// TwinCAT 3 PLC project StringsTests
// ProgramVersion: 3.1.4024.0
// libraries:
//   Strings, * (TomasRompotl)
//   Tc2_Standard, * (Beckhoff Automation GmbH)
//   Tc2_System, * (Beckhoff Automation GmbH)
//   Tc3_Module, * (Beckhoff Automation GmbH)
//   TcUnit, * (www.tcunit.org)
//   Types, * (TomasRompotl)
// project tree:
//   / PlcTask.TcTTO
//   Tests/Builders/ StringBuilder255Test.TcPOU, BuildStringInlineTest.TcPOU, StringBuilderExtBufferTest.TcPOU, StringBuilderInfiniteTest.TcPOU
//   Tests/Convert/ ConvertFunctionsTest.TcPOU
//   Tests/Manipulate/ ManipulateFunctionsTest.TcPOU
//   Tests/ PRG_Test.TcPOU
//   Tests/Validate/ ValidateFunctionsTest.TcPOU
//   Tests/_TemplateTest/ _TemplateTest.TcPOU
// (motion and I/O tree: see PLC project types)
// real-time tasks:
//   TASK BindingTestTask: cycle T#10ms, priority 20, ADS port 350
//   TASK PlcTask: cycle T#10ms, priority 21, ADS port 351
//   TASK PlcTask1: cycle T#10ms, priority 22, ADS port 352
//   TASK PlcTask2: cycle T#10ms, priority 23, ADS port 353

CONFIGURATION StringsTests
    RESOURCE PLC ON TwinCAT3
        TASK PlcTask(INTERVAL := T#1ms, PRIORITY := 21);
        PROGRAM PRG_Test WITH PlcTask : PRG_Test;
    END_RESOURCE
END_CONFIGURATION

// ---- Tests/PRG_Test.TcPOU
PROGRAM PRG_Test
VAR
	validateFunctionsTest : ValidateFunctionsTest;
	manipulateFunctionsTest : ManipulateFunctionsTest;
	convertFunctionsTest : ConvertFunctionsTest;
	
	sb255Test : StringBuilder255Test;
	buildStringInlineTest : BuildStringInlineTest;
	sbExtBufferTest : StringBuilderExtBufferTest;
	sbInfiniteTest : StringBuilderInfiniteTest;
END_VAR

TcUnit.RUN();

END_PROGRAM

// ---- Tests/Validate/ValidateFunctionsTest.TcPOU
FUNCTION_BLOCK ValidateFunctionsTest EXTENDS TcUnit.FB_TestSuite
VAR
END_VAR

StringBeginsWithAnyFunction();
StringEndsWithAnyFunction();
StringBeginsWithFunction();
StringEndsWithFunction();

METHOD StringBeginsWithAnyFunction : BOOL
VAR
	test : T_MaxString := 'this is test string';
END_VAR
TcUnit.TEST('String begins with');

AssertEquals_BOOL(
	Expected := FALSE,
	Actual := StringBeginsWithAny(test, 'nothing'),
	Message := 'Should return FALSE because string does not begin with checked value');

AssertEquals_BOOL(
	Expected := TRUE,
	Actual := StringBeginsWithAny(test, 'this'),
	Message := 'Should return TRUE because string begins with checked value');

TEST_FINISHED();
END_METHOD

METHOD StringBeginsWithFunction
VAR
	test : T_MaxString := 'this is test string';
END_VAR
TcUnit.TEST('String begins with function');

AssertEquals_BOOL(
	Expected := FALSE,
	Actual := StringBeginsWith(test, 'nothing'),
	Message := 'Should return FALSE because string does not begin with checked value');

AssertEquals_BOOL(
	Expected := TRUE,
	Actual := StringBeginsWith(test, 'this'),
	Message := 'Should return TRUE because string begins with checked value');

TEST_FINISHED();
END_METHOD

METHOD StringEndsWithAnyFunction : BOOL
VAR
	test : T_MaxString := 'this is test string';
END_VAR
TcUnit.TEST('String ends with');

AssertEquals_BOOL(
	Expected := FALSE,
	Actual := StringBeginsWithAny(test, 'nothing'),
	Message := 'Should return FALSE because string does not end with checked value');

AssertEquals_BOOL(
	Expected := TRUE,
	Actual := StringEndsWithAny(test, 'string'),
	Message := 'Should return TRUE because string ends with checked value');

TEST_FINISHED();
END_METHOD

METHOD StringEndsWithFunction
VAR
	test : T_MaxString := 'this is test string';
END_VAR
TcUnit.TEST('String ends with function');

AssertEquals_BOOL(
	Expected := FALSE,
	Actual := StringBeginsWith(test, 'nothing'),
	Message := 'Should return FALSE because string does not end with checked value');

AssertEquals_BOOL(
	Expected := TRUE,
	Actual := StringEndsWith(test, 'string'),
	Message := 'Should return TRUE because string ends with checked value');

TEST_FINISHED();
END_METHOD

END_FUNCTION_BLOCK

// ---- Tests/Manipulate/ManipulateFunctionsTest.TcPOU
FUNCTION_BLOCK ManipulateFunctionsTest EXTENDS TcUnit.FB_TestSuite
VAR
END_VAR

AddLeadingZerosFunction();
GetStringBetweenFunction();
RemoveStringFromEndFunction();
ReplaceStringFunction();
ReplaceAllFunction();
ReplaceAllAnyFunction();
ReplaceAllAnyTypeFunction();
SubstringFunction();

METHOD AddLeadingZerosFunction : BOOL
VAR
	test : T_MaxString := '555';
END_VAR
TcUnit.TEST('Add leading zeros');

AssertEquals_STRING(
	Expected := '00555',
	Actual := AddLeadingZeros(test, 5),
	Message := 'Should pad propper number of zeros');

AssertEquals_STRING(
	Expected := '555',
	Actual := AddLeadingZeros(test, 2),
	Message := 'Should do nothing if formatter string already has more chars');

TEST_FINISHED();
END_METHOD

METHOD GetStringBetweenFunction : BOOL
VAR
	test0 : T_MaxString := '1';
	test1 : T_MaxString := '[2]';
	test2 : T_MaxString := 'TestValue[3]rest';
	actual : T_MaxString;
END_VAR
TcUnit.TEST('Get string between');

actual := GetStringBetween(test0, '[', ']');

AssertEquals_STRING(
	Expected := '',
	Actual := actual,
	Message := 'Should return nothing');

actual := GetStringBetween(test1, '[', ']');

AssertEquals_STRING(
	Expected := '2',
	Actual := actual,
	Message := 'Should return content of brackets');

actual := GetStringBetween(test2, '[', ']');

AssertEquals_STRING(
	Expected := '3',
	Actual := actual,
	Message := 'Should return content of brackets');

TEST_FINISHED();
END_METHOD

METHOD RemoveStringFromEndFunction : BOOL
VAR
	test : T_MaxString := 'Last word will be removed';
	actual : T_MaxString;
END_VAR
TcUnit.TEST('Remove string from end function');

actual := RemoveStringFromEnd(test, 'removed');

AssertEquals_STRING(
	Expected := 'Last word will be ',
	Actual := actual,
	Message := 'Should remove last word from test string');

TEST_FINISHED();
END_METHOD

METHOD ReplaceAllAnyFunction
VAR  
	inputString : T_MaxString := 'Valve1 is open';
	substringToReplace : T_MaxString := 'Valve1'; 
	replacementSubstring : T_MaxString := 'Valve2';
 
END_VAR
TcUnit.TEST('Replace all any function');  

ReplaceAllAny(inputString, substringToReplace, replacementSubstring); 

AssertEquals_STRING(
	Expected := 'Valve2 is open',
	Actual := inputString,
	Message := 'Should delete the substring if replacement is empty');
	
TEST_FINISHED();
END_METHOD

METHOD ReplaceAllAnyTypeFunction
VAR  
	inputString  : T_MaxString; 
	substringToReplace : T_MaxString;
	replacementSubstring : T_MaxString;
END_VAR
TcUnit.TEST('Replace all any type function');

inputString  := 'Valve1 is open';
substringToReplace := 'Valve1';
replacementSubstring  := 'Valve2';

ReplaceAllAnyType(ToAnyType(inputString), substringToReplace, replacementSubstring); 

AssertEquals_STRING(
	Expected := 'Valve2 is open',
	Actual := inputString,
	Message := 'ReplaceAllAnyType should delete the substring if replacement is empty');
	
inputString  := 'Valve1 is open';
substringToReplace := 'Valve4';
replacementSubstring  := 'Valve2';

ReplaceAllAnyType(ToAnyType(inputString), substringToReplace, replacementSubstring); 

AssertEquals_STRING(
	Expected := 'Valve1 is open',
	Actual := inputString,
	Message := 'ReplaceAllAnyType should not modify the string if no match is found');
	
inputString  := 'Valve1 is open';
substringToReplace := 'Valve1';
replacementSubstring  := '';

ReplaceAllAnyType(ToAnyType(inputString), substringToReplace, replacementSubstring);

AssertEquals_STRING(
	Expected := ' is open',
	Actual := inputString,
	Message := 'ReplaceAllAnyType should delete the substring if replacement is empty');
	
inputString  := 'Valve1 is open. Valve1 is closed';
substringToReplace := 'Valve1';
replacementSubstring  := 'V1';

ReplaceAllAnyType(ToAnyType(inputString), substringToReplace, replacementSubstring);

AssertEquals_STRING(
	Expected := 'V1 is open. V1 is closed',
	Actual := inputString,
	Message := 'ReplaceAllAnyType should replace all occurrences of the target text');

TEST_FINISHED();
END_METHOD

METHOD ReplaceAllFunction
VAR
	inputString  : T_MaxString;
	substringToReplace : T_MaxString;
	replacementSubstring  : T_MaxString;
END_VAR
TcUnit.TEST('Replace all function');

inputString  := 'Valve1 is open';
substringToReplace := 'Valve1';
replacementSubstring  := 'Valve2';
 
AssertEquals_STRING(
	Expected := 'Valve2 is open',
	Actual := ReplaceAll(inputString, substringToReplace, replacementSubstring),
	Message := 'ReplaceAll should correctly replace the target substring in the input string');
	
inputString  := 'Valve1 is open';
substringToReplace := 'Valve4';
replacementSubstring  := 'Valve2';

AssertEquals_STRING(
	Expected := 'Valve1 is open',
	Actual := ReplaceAll(inputString, substringToReplace, replacementSubstring),
	Message := 'Should not modify the string if no match is found');
	
inputString  := 'Valve1 is open';
substringToReplace := 'Valve1';
replacementSubstring  := '';

AssertEquals_STRING(
	Expected := ' is open',
	Actual := ReplaceAll(inputString, substringToReplace, replacementSubstring),
	Message := 'Should delete the substring if replacement is empty');
	
inputString  := 'Valve1 is open. Valve1 is closed';
substringToReplace := 'Valve1';
replacementSubstring  := 'V1';

AssertEquals_STRING(
	Expected := 'V1 is open. V1 is closed',
	Actual := ReplaceAll(inputString, substringToReplace, replacementSubstring),
	Message := 'ReplaceAll should replace all occurrences of the target text');

TEST_FINISHED();
END_METHOD

METHOD ReplaceStringFunction : BOOL
VAR
	test : T_MaxString := 'this is test string';
END_VAR
TcUnit.TEST('Replace string');

ReplaceString(test, 'not here', 'replaced');

AssertEquals_STRING(
	Expected := 'this is test string',
	Actual := test,
	Message := 'Should do nothing because searched string is not there');

ReplaceString(test, 'test', 'replaced');

AssertEquals_STRING(
	Expected := 'this is replaced string',
	Actual := test,
	Message := 'Should replace found string');

TEST_FINISHED();
END_METHOD

METHOD SubstringFunction
VAR
	source : T_MaxString :=  'ABCDEF123456789';
	destination : T_MaxString;
	startIndex : DINT := 3; 
    length : DINT := 5;	  
END_VAR
TcUnit.TEST('SubString function');

SubString(source, destination, startIndex, length);
AssertEquals_STRING(Expected := 'DEF12',
					Actual :=  destination, 
					Message := 'Substring result incorrect');

TEST_FINISHED();
END_METHOD

END_FUNCTION_BLOCK

// ---- Tests/Convert/ConvertFunctionsTest.TcPOU
FUNCTION_BLOCK ConvertFunctionsTest EXTENDS TcUnit.FB_TestSuite
VAR
END_VAR

AnyToStringFunction();
StringToAnyFunction();

METHOD AnyToStringFunction : BOOL
VAR
	stringVar : T_MaxString := 'test';
	intVar : INT := 42;
	realVar : REAL := 3.14;
END_VAR
TcUnit.TEST('ANY to STRING function');

AssertEquals_STRING(
	Expected := 'test',
	Actual := AnyToString(stringVar),
	Message := 'Should convert STRING var to STRING');

AssertEquals_STRING(
	Expected := '42',
	Actual := AnyToString(intVar),
	Message := 'Should convert INT var to STRING');

AssertEquals_STRING(
	Expected := '3.14',
	Actual := AnyToString(realVar),
	Message := 'Should convert REAL var to STRING');
	
TEST_FINISHED();
END_METHOD

METHOD StringToAnyFunction : BOOL
VAR
	stringVar : T_MaxString;
	intVar : INT;
	realVar : REAL;
END_VAR
TcUnit.TEST('STRING to ANY function');

StringToAny('this is test', stringVar);
StringToAny('42', intVar);
StringToAny('3.14', realVar);

AssertEquals_STRING(
	Expected := 'this is test',
	Actual := stringVar,
	Message := 'Should return correct STRING value');

AssertEquals_INT(
	Expected := 42,
	Actual := intVar,
	Message := 'Should return correct INT value');

AssertEquals_REAL(
	Expected := 3.14,
	Actual := realVar,
	Delta := 0.001,
	Message := 'Should return correct REAL value');

TEST_FINISHED();
END_METHOD

END_FUNCTION_BLOCK

// ---- Tests/Builders/StringBuilder255Test.TcPOU
FUNCTION_BLOCK StringBuilder255Test EXTENDS TcUnit.FB_TestSuite
VAR
END_VAR

AppendAndClear();

METHOD AppendAndClear : BOOL
VAR
	builder : StringBuilder255;
END_VAR
TcUnit.TEST('Append and Clear');

builder
	.Clear()
	.Append('1')
	.Append('2');

AssertEquals_STRING(
	Expected := '12',
	Actual := builder.GetString(),
	Message := 'Should return Appended strings using GetString() method');

AssertEquals_STRING(
	Expected := '12',
	Actual := builder.Value,
	Message := 'Should return string using Value property');

AssertEquals_DINT(
	Expected := 2,
	Actual := builder.Length,
	Message := 'Should return string length');	

builder.Clear();

AssertEquals_BOOL(
	Expected := TRUE,
	Actual := builder.IsEmpty,
	Message := 'Should return that string is empty');
	
TEST_FINISHED();
END_METHOD

END_FUNCTION_BLOCK

// ---- Tests/Builders/BuildStringInlineTest.TcPOU
FUNCTION_BLOCK BuildStringInlineTest EXTENDS TcUnit.FB_TestSuite
VAR
END_VAR

BuildStringInSingleLine();

METHOD BuildStringInSingleLine : BOOL
VAR
END_VAR
TcUnit.TEST('Build string in single line');

AssertEquals_STRING(
	Expected := '12',
	Actual := BuildStringInline('1').Append('2').GetString(),
	Message := 'Should return built string');

AssertEquals_STRING(
	Expected := 'ab',
	Actual := BuildStringInline('a').Append('b').GetString(),
	Message := 'Should return another built string');

TEST_FINISHED();
END_METHOD

END_FUNCTION_BLOCK

// ---- Tests/Builders/StringBuilderExtBufferTest.TcPOU
FUNCTION_BLOCK StringBuilderExtBufferTest EXTENDS TcUnit.FB_TestSuite
VAR
END_VAR

AppendAndClear();

METHOD AppendAndClear : BOOL
VAR
	buffer : STRING(2000);
	builder : StringBuilderExtBuffer := (Buffer := ToAnyType(buffer));
	
	testValue : STRING := ' very long strings';
END_VAR
TcUnit.TEST('Append and Clear');

builder
	.Clear()
	.Append('SB with external buffer')
	.Append(' is meant for')
	.AppendByPointer(ADR(testValue));

AssertEquals_STRING(
	Expected := 'SB with external buffer is meant for very long strings',
	Actual := buffer,
	Message := 'Strings should be properly appended');

builder.Clear();

AssertEquals_BOOL(
	Expected := TRUE,
	Actual := builder.IsEmpty,
	Message := 'Buffer should be empty');
	
TEST_FINISHED();
END_METHOD

END_FUNCTION_BLOCK

// ---- Tests/Builders/StringBuilderInfiniteTest.TcPOU
FUNCTION_BLOCK StringBuilderInfiniteTest EXTENDS TcUnit.FB_TestSuite
VAR
END_VAR

AppendAndClear();
CheckCapacityHasIncreased();

METHOD AppendAndClear : BOOL
VAR
	builder : StringBuilderInfinite;
	testValue : STRING := ' very long strings without care';
END_VAR
TcUnit.TEST('Append and Clear');

builder
	.Clear()
	.Append('SB infinite')
	.Append(' is meant for')
	.AppendByPointer(ADR(testValue));

AssertEquals_STRING(
	Expected := 'SB infinite is meant for very long strings without care',
	Actual := builder.Value^,
	Message := 'Strings should be properly appended');

builder.Clear();

AssertEquals_BOOL(
	Expected := TRUE,
	Actual := builder.IsEmpty,
	Message := 'String should be empty');
	
TEST_FINISHED();
END_METHOD

METHOD CheckCapacityHasIncreased : BOOL
VAR
	builder : StringBuilderInfinite;
	i : INT;
END_VAR
TcUnit.TEST('Check capacity has increased');

AssertEquals_DINT(
	Expected := 1024,
	Actual := builder.Capacity,
	Message := 'Initial capacity should be 1000');
	
builder.Clear();
FOR i := 0 TO 999 DO
	builder.Append('0123456789');
END_FOR

AssertEquals_DINT(
	Expected := 10000,
	Actual := builder.Length,
	Message := 'String should be 10000 long');

AssertEquals_DINT(
	Expected := 16384,
	Actual := builder.Capacity,
	Message := 'Capacity should be increased to 16384');
	
TEST_FINISHED();
END_METHOD

END_FUNCTION_BLOCK

// ---- Tests/_TemplateTest/_TemplateTest.TcPOU
FUNCTION_BLOCK _TemplateTest EXTENDS TcUnit.FB_TestSuite
VAR
END_VAR

ExampleTest();

METHOD ExampleTest : BOOL
VAR
	expected : INT;
	actual : INT;
END_VAR
TcUnit.TEST('Example test');

expected := ;
actual := ;

AssertEquals(
	Expected := expected,
	Actual := actual,
	Message := 'What went wrong');

TEST_FINISHED();
END_METHOD

END_FUNCTION_BLOCK
